// Reserved; prefer Plant or Thread for current code.
FUNCTION_BLOCK SubPlant
VAR
	iFirstCyclic: I_ExecuteNode;
	iLastCyclic: I_ExecuteNode;
	
	iFirstWorker: I_Worker;
	iLastWorker: I_Worker;
END_VAR

METHOD Run
VAR_INPUT
END_VAR
IF _Plant.bInit THEN
	RETURN;
END_IF
END_METHOD

END_FUNCTION_BLOCK

(* stored: Version 1.1.0.1
   POU SubPlant: Id {8b3646af-7c89-4248-ba4b-bde043ef6a9a}, SpecialFunc None
   Method Run: Id {312d03b0-5785-4da7-8eb1-55c23394ad73} *)
